TYPE aT_Turbine :
STRUCT
	Rotation: REAL;
	HighPressure: REAL;
	ImmediatePressure: REAL;
	OutPressure: REAL;
	HighTemperature: REAL;
	ImmediateTemperature: REAL;
	OutTemperature: REAL;
END_STRUCT
END_TYPE

(* stored: Version 1.1.0.1, ProductVersion 3.1.4024.4
   DUT aT_Turbine: Id {f0bb29c6-d156-4be1-9b63-87f431b34ac8} *)
